// TIA Portal V17 export
// export: Created 2025-06-26T06:49:14.0899268Z, ExportSetting WithDefaults, DisplayName Totally Integrated Automation Portal, DisplayVersion V17 Update 8, DisplayName TIA Portal Openness, DisplayVersion V17 Update 8, DisplayName TIA Portal Version Control Interface, DisplayVersion V17, DisplayName STEP 7 Professional, DisplayVersion V17 Update 8, DisplayName STEP 7 Safety, DisplayVersion V17 Update 6, DisplayName WinCC Advanced, DisplayVersion V17 Update 8
FUNCTION_BLOCK "OutputProcessing"   // FB11, FBD
TITLE = Output mapping
{ S7_Optimized_Access := 'TRUE' }
VERSION : 0.1
// stored: AutoNumber true, IsIECCheckEnabled false, IsRetainMemResEnabled false, MemoryReserve 0, SetENOAutomatically false, UDAEnableTagReadback false
BEGIN

REGION Network 1: Digital
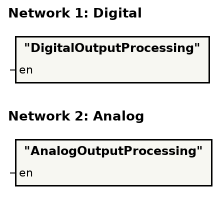
   "DigitalOutputProcessing"();
END_REGION

REGION Network 2: Analog
   "AnalogOutputProcessing"();
END_REGION
END_FUNCTION_BLOCK
